FUNCTION F_CreateStringForCameraProgramNumber : String(10)
VAR_INPUT
	iProgramNumber: UINT;
END_VAR
VAR
	sProgramNumber :STRING(3); //camera number with zeros
END_VAR

// Nullákkal kiegészítés 3 karakterre
IF iProgramNumber < 10 THEN
    sProgramNumber := CONCAT('00', TO_STRING(iProgramNumber));
ELSIF iProgramNumber < 100 THEN
    sProgramNumber := CONCAT('0', TO_STRING(iProgramNumber));
ELSE
    sProgramNumber := TO_STRING(iProgramNumber);
END_IF

// Végső string összeállítása
F_CreateStringForCameraProgramNumber := CONCAT(CONCAT('PW,', sProgramNumber), '$0D');

END_FUNCTION

(* stored: Version 1.1.0.1, ProductVersion 3.1.4024.14
   POU F_CreateStringForCameraProgramNumber: Id {ed3d8e16-360a-40eb-8444-acaf4f9cca61}, SpecialFunc None *)
